# EPICS substitutions: bsaDriverApp/Db/bsss.substitutions
file serviceChannelCtrl.db {
    pattern {   DEVICE,                  DESC,    SERVICE}
            {   "$(DEV)", "$(DESC\=\$\(SECN\))",  "BSSS" }
}

file devBsssScal.db {
    pattern {   IDX,     MDID,   DEVICE,        EGU,        ADEL,        PREC,        HOPR,        LOPR,  DESC  }
#
# user Edefs
#
            {   "0",     "21", "$(DEV)", "$(EGU\=)", "$(ADEL\=)", "$(PREC\=)", "$(HOPR\=)", "$(LOPR\=)", "$(DESC\=\$\(SECN\))" }
            {   "1",     "22", "$(DEV)", "$(EGU\=)", "$(ADEL\=)", "$(PREC\=)", "$(HOPR\=)", "$(LOPR\=)", "$(DESC\=\$\(SECN\))" }
            {   "2",     "23", "$(DEV)", "$(EGU\=)", "$(ADEL\=)", "$(PREC\=)", "$(HOPR\=)", "$(LOPR\=)", "$(DESC\=\$\(SECN\))" }
            {   "3",     "24", "$(DEV)", "$(EGU\=)", "$(ADEL\=)", "$(PREC\=)", "$(HOPR\=)", "$(LOPR\=)", "$(DESC\=\$\(SECN\))" }
            {   "4",     "25", "$(DEV)", "$(EGU\=)", "$(ADEL\=)", "$(PREC\=)", "$(HOPR\=)", "$(LOPR\=)", "$(DESC\=\$\(SECN\))" }
            {   "5",     "26", "$(DEV)", "$(EGU\=)", "$(ADEL\=)", "$(PREC\=)", "$(HOPR\=)", "$(LOPR\=)", "$(DESC\=\$\(SECN\))" }
            {   "6",     "27", "$(DEV)", "$(EGU\=)", "$(ADEL\=)", "$(PREC\=)", "$(HOPR\=)", "$(LOPR\=)", "$(DESC\=\$\(SECN\))" }
            {   "7",     "28", "$(DEV)", "$(EGU\=)", "$(ADEL\=)", "$(PREC\=)", "$(HOPR\=)", "$(LOPR\=)", "$(DESC\=\$\(SECN\))" }
            {   "8",     "29", "$(DEV)", "$(EGU\=)", "$(ADEL\=)", "$(PREC\=)", "$(HOPR\=)", "$(LOPR\=)", "$(DESC\=\$\(SECN\))" }
            {   "9",     "30", "$(DEV)", "$(EGU\=)", "$(ADEL\=)", "$(PREC\=)", "$(HOPR\=)", "$(LOPR\=)", "$(DESC\=\$\(SECN\))" }
#
            {  "10",     "31", "$(DEV)", "$(EGU\=)", "$(ADEL\=)", "$(PREC\=)", "$(HOPR\=)", "$(LOPR\=)", "$(DESC\=\$\(SECN\))" }
            {  "11",     "32", "$(DEV)", "$(EGU\=)", "$(ADEL\=)", "$(PREC\=)", "$(HOPR\=)", "$(LOPR\=)", "$(DESC\=\$\(SECN\))" }
            {  "12",     "33", "$(DEV)", "$(EGU\=)", "$(ADEL\=)", "$(PREC\=)", "$(HOPR\=)", "$(LOPR\=)", "$(DESC\=\$\(SECN\))" }
            {  "13",     "34", "$(DEV)", "$(EGU\=)", "$(ADEL\=)", "$(PREC\=)", "$(HOPR\=)", "$(LOPR\=)", "$(DESC\=\$\(SECN\))" }
            {  "14",     "35", "$(DEV)", "$(EGU\=)", "$(ADEL\=)", "$(PREC\=)", "$(HOPR\=)", "$(LOPR\=)", "$(DESC\=\$\(SECN\))" }
            {  "15",     "36", "$(DEV)", "$(EGU\=)", "$(ADEL\=)", "$(PREC\=)", "$(HOPR\=)", "$(LOPR\=)", "$(DESC\=\$\(SECN\))" }
            {  "16",     "37", "$(DEV)", "$(EGU\=)", "$(ADEL\=)", "$(PREC\=)", "$(HOPR\=)", "$(LOPR\=)", "$(DESC\=\$\(SECN\))" }
            {  "17",     "38", "$(DEV)", "$(EGU\=)", "$(ADEL\=)", "$(PREC\=)", "$(HOPR\=)", "$(LOPR\=)", "$(DESC\=\$\(SECN\))" }
            {  "18",     "39", "$(DEV)", "$(EGU\=)", "$(ADEL\=)", "$(PREC\=)", "$(HOPR\=)", "$(LOPR\=)", "$(DESC\=\$\(SECN\))" }
            {  "19",     "40", "$(DEV)", "$(EGU\=)", "$(ADEL\=)", "$(PREC\=)", "$(HOPR\=)", "$(LOPR\=)", "$(DESC\=\$\(SECN\))" }
#
            {  "20",     "41", "$(DEV)", "$(EGU\=)", "$(ADEL\=)", "$(PREC\=)", "$(HOPR\=)", "$(LOPR\=)", "$(DESC\=\$\(SECN\))" }
            {  "21",     "42", "$(DEV)", "$(EGU\=)", "$(ADEL\=)", "$(PREC\=)", "$(HOPR\=)", "$(LOPR\=)", "$(DESC\=\$\(SECN\))" }
            {  "22",     "43", "$(DEV)", "$(EGU\=)", "$(ADEL\=)", "$(PREC\=)", "$(HOPR\=)", "$(LOPR\=)", "$(DESC\=\$\(SECN\))" }
            {  "23",     "44", "$(DEV)", "$(EGU\=)", "$(ADEL\=)", "$(PREC\=)", "$(HOPR\=)", "$(LOPR\=)", "$(DESC\=\$\(SECN\))" }
            {  "24",     "45", "$(DEV)", "$(EGU\=)", "$(ADEL\=)", "$(PREC\=)", "$(HOPR\=)", "$(LOPR\=)", "$(DESC\=\$\(SECN\))" }
            {  "25",     "46", "$(DEV)", "$(EGU\=)", "$(ADEL\=)", "$(PREC\=)", "$(HOPR\=)", "$(LOPR\=)", "$(DESC\=\$\(SECN\))" }
            {  "26",     "47", "$(DEV)", "$(EGU\=)", "$(ADEL\=)", "$(PREC\=)", "$(HOPR\=)", "$(LOPR\=)", "$(DESC\=\$\(SECN\))" }
            {  "27",     "48", "$(DEV)", "$(EGU\=)", "$(ADEL\=)", "$(PREC\=)", "$(HOPR\=)", "$(LOPR\=)", "$(DESC\=\$\(SECN\))" }
            {  "28",     "49", "$(DEV)", "$(EGU\=)", "$(ADEL\=)", "$(PREC\=)", "$(HOPR\=)", "$(LOPR\=)", "$(DESC\=\$\(SECN\))" }
#
# system Edefs
#
            {  "29",  "SCD1H", "$(DEV)", "$(EGU\=)", "$(ADEL\=)", "$(PREC\=)", "$(HOPR\=)", "$(LOPR\=)", "$(DESC\=\$\(SECN\))" }
            {  "30",  "SCDTH", "$(DEV)", "$(EGU\=)", "$(ADEL\=)", "$(PREC\=)", "$(HOPR\=)", "$(LOPR\=)", "$(DESC\=\$\(SECN\))" }
            {  "31",  "SCDHH", "$(DEV)", "$(EGU\=)", "$(ADEL\=)", "$(PREC\=)", "$(HOPR\=)", "$(LOPR\=)", "$(DESC\=\$\(SECN\))" }
            {  "32",  "SCL1H", "$(DEV)", "$(EGU\=)", "$(ADEL\=)", "$(PREC\=)", "$(HOPR\=)", "$(LOPR\=)", "$(DESC\=\$\(SECN\))" }
            {  "33",  "SCLTH", "$(DEV)", "$(EGU\=)", "$(ADEL\=)", "$(PREC\=)", "$(HOPR\=)", "$(LOPR\=)", "$(DESC\=\$\(SECN\))" }
            {  "34",  "SCLHH", "$(DEV)", "$(EGU\=)", "$(ADEL\=)", "$(PREC\=)", "$(HOPR\=)", "$(LOPR\=)", "$(DESC\=\$\(SECN\))" }
            {  "35",  "SCB1H", "$(DEV)", "$(EGU\=)", "$(ADEL\=)", "$(PREC\=)", "$(HOPR\=)", "$(LOPR\=)", "$(DESC\=\$\(SECN\))" }
            {  "36",  "SCBTH", "$(DEV)", "$(EGU\=)", "$(ADEL\=)", "$(PREC\=)", "$(HOPR\=)", "$(LOPR\=)", "$(DESC\=\$\(SECN\))" }
            {  "37",  "SCBHH", "$(DEV)", "$(EGU\=)", "$(ADEL\=)", "$(PREC\=)", "$(HOPR\=)", "$(LOPR\=)", "$(DESC\=\$\(SECN\))" }
            {  "38",  "SCH1H", "$(DEV)", "$(EGU\=)", "$(ADEL\=)", "$(PREC\=)", "$(HOPR\=)", "$(LOPR\=)", "$(DESC\=\$\(SECN\))" }
            {  "39",  "SCHTH", "$(DEV)", "$(EGU\=)", "$(ADEL\=)", "$(PREC\=)", "$(HOPR\=)", "$(LOPR\=)", "$(DESC\=\$\(SECN\))" }
            {  "40",  "SCHHH", "$(DEV)", "$(EGU\=)", "$(ADEL\=)", "$(PREC\=)", "$(HOPR\=)", "$(LOPR\=)", "$(DESC\=\$\(SECN\))" }
            {  "41",  "SCS1H", "$(DEV)", "$(EGU\=)", "$(ADEL\=)", "$(PREC\=)", "$(HOPR\=)", "$(LOPR\=)", "$(DESC\=\$\(SECN\))" }
            {  "42",  "SCSTH", "$(DEV)", "$(EGU\=)", "$(ADEL\=)", "$(PREC\=)", "$(HOPR\=)", "$(LOPR\=)", "$(DESC\=\$\(SECN\))" }
            {  "43",  "SCSHH", "$(DEV)", "$(EGU\=)", "$(ADEL\=)", "$(PREC\=)", "$(HOPR\=)", "$(LOPR\=)", "$(DESC\=\$\(SECN\))" }
}
